TYPE TYP_REAL_XYZ :
STRUCT
	X : REAL;
	Y : REAL;
	Z : REAL;
END_STRUCT
END_TYPE

(* stored: Version 1.1.0.1, ProductVersion 3.1.4024.12
   DUT TYP_REAL_XYZ: Id {09a4efa0-8aa0-41a0-a17f-4c95f853bd1d} *)
